FUNCTION_BLOCK FB_Display IMPLEMENTS IDisplay
VAR
END_VAR

METHOD Show : BOOL
VAR_INPUT
	Message : T_MaxString;
END_VAR
ADSLOGSTR(msgCtrlMask := ADSLOG_MSGTYPE_LOG, msgFmtStr := '%s', strArg := Message);
END_METHOD

END_FUNCTION_BLOCK

(* stored: Version 1.1.0.1, ProductVersion 3.1.4024.12
   POU FB_Display: Id {0f56468b-8a03-496b-85ad-d04670cb0ef2}, SpecialFunc None
   Method Show: Id {5434fd17-59a5-4839-a6dc-4e3706325968} *)
